KUKA KRL program: second_plfs_select.src, second_plfs_select.dat

--- second_plfs_select.src ---
&ACCESS RV
&REL 1
&PARAM DISKPATH = KRC:\R1\Program\SecondSortMain
&comment Plfs Select
def second_plfs_select()
;***********************************************************
;
; Copyright 2018 - 2024 speedbot All Rights reserved.
;
; File Name: second_plfs_select.src
;
; Description:
;   Language             ==   Krl for KUKA ROBOT
;   Date                 ==   2022 - 06 - 27
;   Modification Data    ==   2024 - 10 - 25
;
; Author: speedbot
;
; Version: 1.1
;***********************************************************

    switch (GlbPartData.BoxId)
    case 1
        second_place01()
    case 2
        second_place02()
    case 3
        second_place03()
    case 4
        second_place04()
    case 5
        second_place05()
    case 6
        second_place06()
    case 7
        second_place07()
    case 8
        second_place08()
    case 9
        second_place09()
    case 10
        second_place10()
    case 11
        second_place11()
    case 12
        second_place12()
    default
        Offset = 0
        swrite(Msg[], State, Offset, "BoxId Error[BoxId:%D, MaxBoxId:%D]", GlbPartData.BoxId, PkPlCfg.NumOfBox)
        err_write_("SecondSort", Msg[], true)
    endswitch
end

--- second_plfs_select.dat ---
&ACCESS RV
&REL 1
&PARAM DISKPATH = KRC:\R1\Program\SecondSortMain
&comment Plfs Select
defdat second_plfs_select
;***********************************************************
;
; Copyright 2018 - 2024 speedbot All Rights reserved.
;
; File Name: second_plfs_select.dat
;
; Description:
;   Language             ==   Krl for KUKA ROBOT
;   Date                 ==   2022 - 06 - 28
;   Modification Data    ==   2022 - 06 - 28
;
; Author: speedbot
;
; Version: 1.0
;***********************************************************

ext second_place01()
ext second_place02()
ext second_place03()
ext second_place04()
ext second_place05()
ext second_place06()
ext second_place07()
ext second_place08()
ext second_place09()
ext second_place10()
ext second_place11()
ext second_place12()

decl state_t State
decl int Offset = 0
decl char Msg[256]

enddat
